FUNCTION_BLOCK AND_EVENTS_bkp (* Basic Function Block Type *)
  (* Standard: 61499-2 *)
  (* Version 0.0, 10/19/2017, chivdan, nxtControl GmbH, Template *)
  PACKAGE Main;
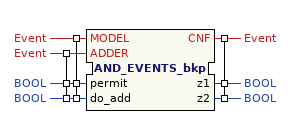
  EVENT_INPUT
    MODEL WITH permit, do_add; (* Normal Execution Request *)
    ADDER WITH permit, do_add;
  END_EVENT
  EVENT_OUTPUT
    CNF WITH z1, z2; (* Execution Confirmation *)
  END_EVENT
  VAR_INPUT
    permit : BOOL;
    do_add : BOOL;
  END_VAR
  VAR_OUTPUT
    z1 : BOOL;
    z2 : BOOL;
  END_VAR
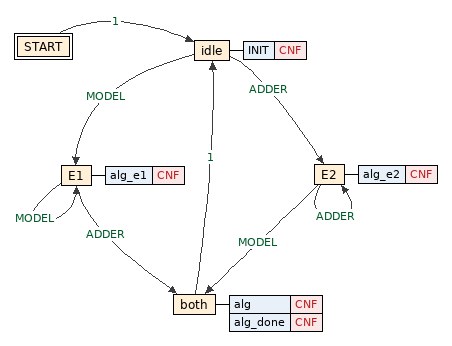
  EC_STATES
    START; (* Initial State *)
    idle : INIT -> CNF; (* Initialization *)
    E1 : alg_e1 -> CNF;
    E2 : alg_e2 -> CNF;
    both : alg -> CNF, alg_done -> CNF;
  END_STATES
  EC_TRANSITIONS
    START TO idle := 1;
    idle TO E1 := MODEL;
    idle TO E2 := ADDER;
    E1 TO both := ADDER;
    E2 TO both := MODEL;
    both TO idle := 1;
    E1 TO E1 := MODEL;
    E2 TO E2 := ADDER;
  END_TRANSITIONS
  ALGORITHM INIT IN ST: (* Initialization algorithm *)
z1:=FALSE;
z2:=FALSE;
MODEL:=FALSE;
ADDER:=FALSE;
  END_ALGORITHM
  ALGORITHM alg_e1 IN ST:
	z1:=permit;



	z2:=do_add;


MODEL:=FALSE;
  END_ALGORITHM
  ALGORITHM alg_done IN ST:
z1:=FALSE;
z2:=FALSE;
MODEL:=FALSE;
ADDER:=FALSE;
  END_ALGORITHM
  ALGORITHM alg_e2 IN ST:
	z1:=permit;



	z2:=do_add;


ADDER:=FALSE;
  END_ALGORITHM
  ALGORITHM alg IN ST:
;

	z1:=permit;



	z2:=do_add;

MODEL:=FALSE;
ADDER:=FALSE;
  END_ALGORITHM
END_FUNCTION_BLOCK
